SUBAPPLICATION SubApp_PC_B (* Geraet B (Station 12, 192.168.1.12): reine SR-Flipflop-Logik (ASR_AX_SR_2, kein Toggle) und DigitalOutput_Q1 - 'SUB style', das Protokoll steckt im MyLib::sys-Composite (SoftKeySR_PC_B_OPC_Adapter), nicht in der Resource des Geraets - Adapter-Variante von Training_05, gleiche OPC-UA-Adressen *)
  (* Standard: 61499-2; Description: Copyright (c) 2026 Meisterschulen am Ostbahnhof This program and the accompanying materials are made available under the terms of the Eclipse Public License 2.0 which is available at https://www.eclipse.org/legal/epl-2.0/ SPDX-License-Identifier: EPL-2.0 *)
  (* Version 1.0, 2026-09-04, Franz Höpfinger, Meisterschulen am Ostbahnhof, initial API and implementation and/or initial documentation *)
  PACKAGE subapp::Training_07_OPC_UA_RES;
  IMPORT logiBUS::io::DQ::logiBUS_DO::Output_Q1;
  IMPORT VV::const::OPC_UA::myOpcUaAddresses::SR2_SET_LOCAL_METHOD;
  IMPORT VV::const::OPC_UA::myOpcUaAddresses::SR2_RESET_LOCAL_METHOD;
  IMPORT VV::const::OPC_UA::myOpcUaAddresses::SR2_STATE_REMOTE_WRITE;
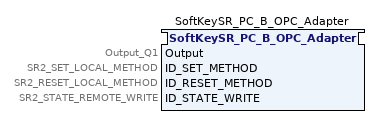
  SUBAPPS
    SoftKeySR_PC_B_OPC_Adapter : MyLib::sys::SoftKeySR_PC_B_OPC_Adapter(Output := Output_Q1, ID_SET_METHOD := SR2_SET_LOCAL_METHOD, ID_RESET_METHOD := SR2_RESET_LOCAL_METHOD, ID_STATE_WRITE := SR2_STATE_REMOTE_WRITE);
  END_SUBAPPS
END_SUBAPPLICATION
